INTERFACE I_Cycle EXTENDS I_Object

END_INTERFACE

(* stored: Version 1.1.0.1
   Itf I_Cycle: Id {e1e2ff06-3bf6-45ba-91e5-14895b5625fb} *)
